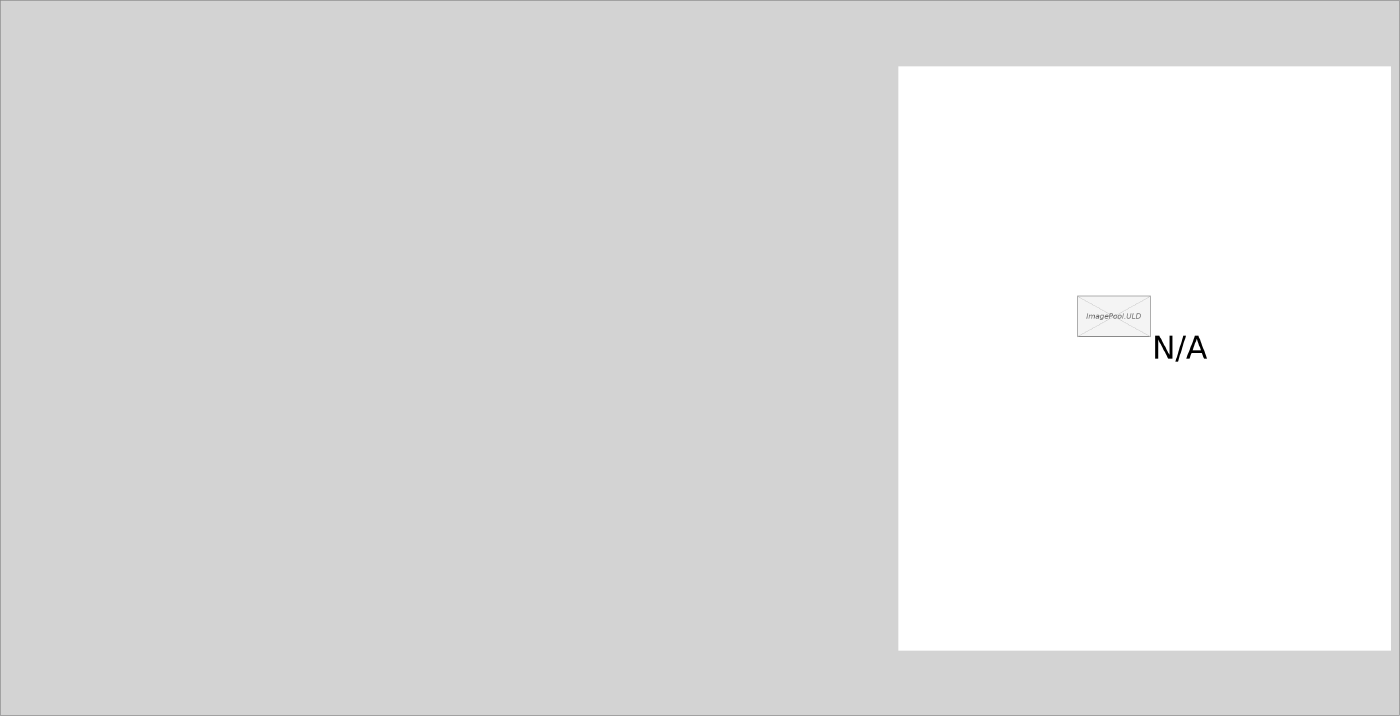
VISUALIZATION Manual_Unloading  // 1920x983
    Rectangle (0,0 1920x983)
    Rectangle (1232,91 675x802)
    Image (1477,406 101x56), image: ImagePool.ULD
    Label (1410,401 416x153), "N/A"
END_VISUALIZATION

(* stored: Version 1.1.0.1, ProductVersion 3.1.4024.12
   Visu Manual_Unloading: Id {ad2805ff-8961-416c-8297-7957208feb8e} *)
